LIN {X 0,Y 105.077,Z 582.031,A -85,B 0,C 180,E1 -30092.346,E2 -30092.346} C_VEL
LIN {X 0,Y 107.471,Z 573.639,A -85,B 0,C 180,E1 -30085.983,E2 -30085.983} C_VEL
LIN {X 0,Y 110.24,Z 565.564,A -85,B 0,C 180,E1 -30081.011,E2 -30081.011} C_VEL
LIN {X 0,Y 113.116,Z 557.316,A -85,B 0,C 180,E1 -30076.748,E2 -30076.748} C_VEL
LIN {X 0,Y 115.626,Z 549.926,A -85,B 0,C 180,E1 -30073.463,E2 -30073.463} C_VEL
LIN {X 0,Y 116.51,Z 546.107,A -85,B 0,C 180,E1 -30071.392,E2 -30071.392} C_VEL
LIN {X 0,Y 117.304,Z 542.305,A -85,B 0,C 180,E1 -30068.612,E2 -30068.612} C_VEL
LIN {X 0,Y 117.606,Z 540.558,A -85,B 0,C 180,E1 -30066.862,E2 -30066.862} C_VEL
LIN {X 0,Y 117.834,Z 538.313,A -85,B 0,C 180,E1 -30063.417,E2 -30063.417} C_VEL
LIN {X 0,Y 118.164,Z 536.971,A -85,B 0,C 180,E1 -30059.786,E2 -30059.786} C_VEL
LIN {X 0,Y 117.435,Z 539.078,A -85,B 0,C 180,E1 -30059.619,E2 -30059.619} C_VEL
LIN {X 0,Y 111.577,Z 552.371,A -85,B 0,C 180,E1 -30059.383,E2 -30059.383} C_VEL
LIN {X 0,Y 105.436,Z 562.957,A -85,B 0,C 180,E1 -30059.029,E2 -30059.029} C_VEL
LIN {X 0,Y 99.299,Z 571.677,A -85,B 0,C 180,E1 -30058.64,E2 -30058.64} C_VEL
LIN {X 0,Y 93.169,Z 579.093,A -85,B 0,C 180,E1 -30058.17,E2 -30058.17} C_VEL
LIN {X 0,Y 84.425,Z 587.882,A -85,B 0,C 180,E1 -30057.383,E2 -30057.383} C_VEL
LIN {X 0,Y 77.446,Z 593.868,A -85,B 0,C 180,E1 -30056.59,E2 -30056.59} C_VEL
LIN {X 0,Y 68.748,Z 600.175,A -85,B 0,C 180,E1 -30055.373,E2 -30055.373} C_VEL
LIN {X 0,Y 59.766,Z 605.63,A -85,B 0,C 180,E1 -30053.555,E2 -30053.555} C_VEL
LIN {X 0,Y 49.832,Z 610.547,A -85,B 0,C 180,E1 -30050.847,E2 -30050.847} C_VEL
LIN {X 0,Y 39.701,Z 614.514,A -85,B 0,C 180,E1 -30046.82,E2 -30046.82} C_VEL
LIN {X 0,Y 29.883,Z 617.454,A -85,B 0,C 180,E1 -30040.186,E2 -30040.186} C_VEL
LIN {X 0,Y 23.761,Z 618.964,A -85,B 0,C 180,E1 -30032.551,E2 -30032.551} C_VEL
LIN {X 0,Y 14.253,Z 620.512,A -85,B 0,C 180,E1 -29999.553,E2 -29999.553} C_VEL
LIN {X 0,Y 12.872,Z 620.802,A -85,B 0,C 180,E1 -29970.009,E2 -29970.009} C_VEL
LIN {X 0,Y 18.308,Z 619.905,A -85,B 0,C 180,E1 -29919.86,E2 -29919.86} C_VEL
LIN {X 0,Y 23.759,Z 618.965,A -85,B 0,C 180,E1 -29907.463,E2 -29907.463} C_VEL
LIN {X 0,Y 36.38,Z 615.606,A -85,B 0,C 180,E1 -29895.017,E2 -29895.017} C_VEL
LIN {X 0,Y 46.424,Z 611.976,A -85,B 0,C 180,E1 -29890.275,E2 -29890.275} C_VEL
LIN {X 0,Y 54.798,Z 608.214,A -85,B 0,C 180,E1 -29887.618,E2 -29887.618} C_VEL
LIN {X 0,Y 65.275,Z 602.361,A -85,B 0,C 180,E1 -29885.202,E2 -29885.202} C_VEL
LIN {X 0,Y 73.957,Z 596.492,A -85,B 0,C 180,E1 -29883.84,E2 -29883.84} C_VEL
LIN {X 0,Y 80.928,Z 591.003,A -85,B 0,C 180,E1 -29882.97,E2 -29882.97} C_VEL
LIN {X 0,Y 89.662,Z 582.792,A -85,B 0,C 180,E1 -29882.072,E2 -29882.072} C_VEL
LIN {X 0,Y 96.667,Z 574.974,A -85,B 0,C 180,E1 -29881.544,E2 -29881.544} C_VEL
LIN {X 0,Y 102.802,Z 566.899,A -85,B 0,C 180,E1 -29881.148,E2 -29881.148} C_VEL
LIN {X 0,Y 108.941,Z 557.148,A -85,B 0,C 180,E1 -29880.804,E2 -29880.804} C_VEL
LIN {X 0,Y 113.845,Z 547.604,A -85,B 0,C 180,E1 -29880.518,E2 -29880.518} C_VEL
LIN {X 0,Y 117.948,Z 537.604,A -85,B 0,C 180,E1 -29880.345,E2 -29880.345} C_VEL
LIN {X 0,Y 118.156,Z 536.995,A -85,B 0,C 180,E1 -29880.214,E2 -29880.214} C_VEL
LIN {X 0,Y 117.764,Z 538.933,A -85,B 0,C 180,E1 -29875.407,E2 -29875.407} C_VEL
LIN {X 0,Y 117.595,Z 540.587,A -85,B 0,C 180,E1 -29873.137,E2 -29873.137} C_VEL
LIN {X 0,Y 117.104,Z 543.335,A -85,B 0,C 180,E1 -29870.502,E2 -29870.502} C_VEL
LIN {X 0,Y 116.14,Z 547.81,A -85,B 0,C 180,E1 -29867.597,E2 -29867.597} C_VEL
LIN {X 0,Y 114.656,Z 552.807,A -85,B 0,C 180,E1 -29865.226,E2 -29865.226} C_VEL
LIN {X 0,Y 111.526,Z 561.914,A -85,B 0,C 180,E1 -29860.948,E2 -29860.948} C_VEL
LIN {X 0,Y 108.525,Z 570.445,A -85,B 0,C 180,E1 -29856.127,E2 -29856.127} C_VEL
LIN {X 0,Y 105.997,Z 578.44,A -85,B 0,C 180,E1 -29850.552,E2 -29850.552} C_VEL
LIN {X 0,Y 104.537,Z 584.513,A -85,B 0,C 180,E1 -29845.536,E2 -29845.536} C_VEL
LIN {X 0,Y 103.789,Z 592.504,A -85,B 0,C 180,E1 -29837.382,E2 -29837.382} C_VEL
LIN {X 0,Y 104.447,Z 596.825,A -85,B 0,C 180,E1 -29832.258,E2 -29832.258} C_VEL
LIN {X 0,Y 106.982,Z 602.173,A -85,B 0,C 180,E1 -29824.805,E2 -29824.805} C_VEL
LIN {X 0,Y 112.946,Z 607.538,A -85,B 0,C 180,E1 -29815.82,E2 -29815.82} C_VEL
LIN {X 0,Y 119.388,Z 610.725,A -85,B 0,C 180,E1 -29809.638,E2 -29809.638} C_VEL
LIN {X 0,Y 130.261,Z 613.684,A -85,B 0,C 180,E1 -29802.462,E2 -29802.462} C_VEL
LIN {X 0,Y 141.664,Z 615.261,A -85,B 0,C 180,E1 -29797.173,E2 -29797.173} C_VEL
LIN {X 0,Y 154.948,Z 615.935,A -85,B 0,C 180,E1 -29792.599,E2 -29792.599} C_VEL
LIN {X 0,Y 164.361,Z 615.933,A -85,B 0,C 180,E1 -29789.999,E2 -29789.999} C_VEL
LIN {X 0,Y 146.045,Z 615.598,A -85,B 0,C 180,E1 -29784.476,E2 -29784.476} C_VEL
LIN {X 0,Y 135.511,Z 614.596,A -85,B 0,C 180,E1 -29780.186,E2 -29780.186} C_VEL
LIN {X 0,Y 128.24,Z 613.248,A -85,B 0,C 180,E1 -29776.399,E2 -29776.399} C_VEL
LIN {X 0,Y 124.259,Z 612.62,A -85,B 0,C 180,E1 -29774.437,E2 -29774.437} C_VEL
LIN {X 0,Y 110.941,Z 610.999,A -85,B 0,C 180,E1 -29768.696,E2 -29768.696} C_VEL
LIN {X 0,Y 107.457,Z 610.024,A -85,B 0,C 180,E1 -29766.262,E2 -29766.262} C_VEL
LIN {X 0,Y 106.575,Z 609.586,A -85,B 0,C 180,E1 -29765.354,E2 -29765.354} C_VEL
LIN {X 0,Y 102.211,Z 606.637,A -85,B 0,C 180,E1 -29759.256,E2 -29759.256} C_VEL
LIN {X 0,Y 98.452,Z 601.21,A -85,B 0,C 180,E1 -29750.023,E2 -29750.023} C_VEL
LIN {X 0,Y 97.503,Z 596.13,A -85,B 0,C 180,E1 -29742.705,E2 -29742.705} C_VEL
LIN {X 0,Y 98.308,Z 589.496,A -85,B 0,C 180,E1 -29734.881,E2 -29734.881} C_VEL
LIN {X 0,Y 100.536,Z 582.409,A -85,B 0,C 180,E1 -29728.151,E2 -29728.151} C_VEL
LIN {X 0,Y 103.813,Z 574.191,A -85,B 0,C 180,E1 -29721.856,E2 -29721.856} C_VEL
LIN {X 0,Y 107.554,Z 565.572,A -85,B 0,C 180,E1 -29716.609,E2 -29716.609} C_VEL
LIN {X 0,Y 111.41,Z 556.493,A -85,B 0,C 180,E1 -29712.154,E2 -29712.154} C_VEL
LIN {X 0,Y 112.579,Z 553.533,A -85,B 0,C 180,E1 -29710.792,E2 -29710.792} C_VEL
LIN {X 0,Y 113.773,Z 550.19,A -85,B 0,C 180,E1 -29708.751,E2 -29708.751} C_VEL
LIN {X 0,Y 114.358,Z 547.971,A -85,B 0,C 180,E1 -29707.058,E2 -29707.058} C_VEL
LIN {X 0,Y 114.767,Z 546.299,A -85,B 0,C 180,E1 -29705.268,E2 -29705.268} C_VEL
LIN {X 0,Y 115.054,Z 545.147,A -85,B 0,C 180,E1 -29703.5,E2 -29703.5} C_VEL
LIN {X 0,Y 114.199,Z 546.967,A -85,B 0,C 180,E1 -29703.047,E2 -29703.047} C_VEL
LIN {X 0,Y 109.078,Z 556.945,A -85,B 0,C 180,E1 -29702.933,E2 -29702.933} C_VEL
LIN {X 0,Y 102.91,Z 566.698,A -85,B 0,C 180,E1 -29702.821,E2 -29702.821} C_VEL
LIN {X 0,Y 94.979,Z 576.963,A -85,B 0,C 180,E1 -29702.628,E2 -29702.628} C_VEL
LIN {X 0,Y 86.163,Z 586.127,A -85,B 0,C 180,E1 -29702.287,E2 -29702.287} C_VEL
LIN {X 0,Y 77.35,Z 593.672,A -85,B 0,C 180,E1 -29701.859,E2 -29701.859} C_VEL
LIN {X 0,Y 68.542,Z 599.979,A -85,B 0,C 180,E1 -29701.314,E2 -29701.314} C_VEL
LIN {X 0,Y 59.742,Z 605.253,A -85,B 0,C 180,E1 -29700.493,E2 -29700.493} C_VEL
LIN {X 0,Y 49.204,Z 610.351,A -85,B 0,C 180,E1 -29699.077,E2 -29699.077} C_VEL
LIN {X 0,Y 38.703,Z 614.318,A -85,B 0,C 180,E1 -29697.167,E2 -29697.167} C_VEL
LIN {X 0,Y 28.274,Z 617.258,A -85,B 0,C 180,E1 -29693.896,E2 -29693.896} C_VEL
LIN {X 0,Y 21.426,Z 618.768,A -85,B 0,C 180,E1 -29689.771,E2 -29689.771} C_VEL
LIN {X 0,Y 8.797,Z 620.316,A -85,B 0,C 180,E1 -29663.046,E2 -29663.046} C_VEL
LIN {X 0,Y 5.76,Z 620.606,A -85,B 0,C 180,E1 -29610.021,E2 -29610.021} C_VEL
LIN {X 0,Y 14.789,Z 619.709,A -85,B 0,C 180,E1 -29538.142,E2 -29538.142} C_VEL
LIN {X 0,Y 21.423,Z 618.769,A -85,B 0,C 180,E1 -29530.243,E2 -29530.243} C_VEL
LIN {X 0,Y 35.213,Z 615.41,A -85,B 0,C 180,E1 -29523.759,E2 -29523.759} C_VEL
LIN {X 0,Y 45.694,Z 611.781,A -85,B 0,C 180,E1 -29521.46,E2 -29521.46} C_VEL
LIN {X 0,Y 56.221,Z 607.046,A -85,B 0,C 180,E1 -29519.891,E2 -29519.891} C_VEL
LIN {X 0,Y 66.778,Z 601.073,A -85,B 0,C 180,E1 -29518.785,E2 -29518.785} C_VEL
LIN {X 0,Y 75.586,Z 594.984,A -85,B 0,C 180,E1 -29518.188,E2 -29518.188} C_VEL
LIN {X 0,Y 82.634,Z 589.249,A -85,B 0,C 180,E1 -29517.849,E2 -29517.849} C_VEL
LIN {X 0,Y 89.687,Z 582.597,A -85,B 0,C 180,E1 -29517.53,E2 -29517.53} C_VEL
LIN {X 0,Y 96.736,Z 574.78,A -85,B 0,C 180,E1 -29517.338,E2 -29517.338} C_VEL
LIN {X 0,Y 102.905,Z 566.704,A -85,B 0,C 180,E1 -29517.189,E2 -29517.189} C_VEL
LIN {X 0,Y 109.072,Z 556.953,A -85,B 0,C 180,E1 -29517.076,E2 -29517.076} C_VEL
LIN {X 0,Y 114.158,Z 547.059,A -85,B 0,C 180,E1 -29516.952,E2 -29516.952} C_VEL
LIN {X 0,Y 115.07,Z 545.112,A -85,B 0,C 180,E1 -29516.5,E2 -29516.5} C_VEL
LIN {X 0,Y 114.759,Z 546.317,A -85,B 0,C 180,E1 -29514.731,E2 -29514.731} C_VEL
LIN {X 0,Y 114.117,Z 548.954,A -85,B 0,C 180,E1 -29512.089,E2 -29512.089} C_VEL
LIN {X 0,Y 112.59,Z 553.513,A -85,B 0,C 180,E1 -29509.209,E2 -29509.209} C_VEL
LIN {X 0,Y 108.961,Z 562.356,A -85,B 0,C 180,E1 -29505.051,E2 -29505.051} C_VEL
LIN {X 0,Y 105.384,Z 570.543,A -85,B 0,C 180,E1 -29500.524,E2 -29500.524} C_VEL
LIN {X 0,Y 102.338,Z 577.72,A -85,B 0,C 180,E1 -29495.669,E2 -29495.669} C_VEL
LIN {X 0,Y 99.681,Z 584.762,A -85,B 0,C 180,E1 -29489.842,E2 -29489.842} C_VEL
LIN {X 0,Y 97.81,Z 592.098,A -85,B 0,C 180,E1 -29482.219,E2 -29482.219} C_VEL
LIN {X 0,Y 97.691,Z 598.503,A -85,B 0,C 180,E1 -29473.998,E2 -29473.998} C_VEL
LIN {X 0,Y 99.573,Z 603.51,A -85,B 0,C 180,E1 -29466.232,E2 -29466.232} C_VEL
LIN {X 0,Y 103.762,Z 607.822,A -85,B 0,C 180,E1 -29458.301,E2 -29458.301} C_VEL
LIN {X 0,Y 108.038,Z 610.419,A -85,B 0,C 180,E1 -29452.972,E2 -29452.972} C_VEL
LIN {X 0,Y 116.685,Z 613.42,A -85,B 0,C 180,E1 -29445.496,E2 -29445.496} C_VEL
LIN {X 0,Y 128.033,Z 615.375,A -85,B 0,C 180,E1 -29438.878,E2 -29438.878} C_VEL
LIN {X 0,Y 143.113,Z 616.254,A -85,B 0,C 180,E1 -29432.814,E2 -29432.814} C_VEL
LIN {X 0,Y 152.408,Z 616.261,A -85,B 0,C 180,E1 -29429.999,E2 -29429.999} C_VEL
LIN {X 0,Y 140.833,Z 616.242,A -85,B 0,C 180,E1 -29426.403,E2 -29426.403} C_VEL
LIN {X 0,Y 126.578,Z 615.235,A -85,B 0,C 180,E1 -29420.411,E2 -29420.411} C_VEL
LIN {X 0,Y 116.686,Z 613.419,A -85,B 0,C 180,E1 -29414.503,E2 -29414.503} C_VEL
LIN {X 0,Y 106.575,Z 609.586,A -85,B 0,C 180,E1 -29405.354,E2 -29405.354} C_VEL
LIN {X 0,Y 103.743,Z 608.404,A -85,B 0,C 180,E1 -29402.603,E2 -29402.603} C_VEL
LIN {X 0,Y 94.034,Z 605.542,A -85,B 0,C 180,E1 -29394.078,E2 -29394.078} C_VEL
LIN {X 0,Y 92.077,Z 604.091,A -85,B 0,C 180,E1 -29390.778,E2 -29390.778} C_VEL
LIN {X 0,Y 91.753,Z 603.497,A -85,B 0,C 180,E1 -29389.63,E2 -29389.63} C_VEL
LIN {X 0,Y 91.292,Z 597.32,A -85,B 0,C 180,E1 -29379.659,E2 -29379.659} C_VEL
LIN {X 0,Y 93.298,Z 590.008,A -85,B 0,C 180,E1 -29370.557,E2 -29370.557} C_VEL
LIN {X 0,Y 96.591,Z 582.776,A -85,B 0,C 180,E1 -29363.585,E2 -29363.585} C_VEL
LIN {X 0,Y 100.516,Z 575.187,A -85,B 0,C 180,E1 -29357.754,E2 -29357.754} C_VEL
LIN {X 0,Y 104.996,Z 566.701,A -85,B 0,C 180,E1 -29352.635,E2 -29352.635} C_VEL
LIN {X 0,Y 109.261,Z 558.245,A -85,B 0,C 180,E1 -29348.527,E2 -29348.527} C_VEL
LIN {X 0,Y 110.195,Z 556.06,A -85,B 0,C 180,E1 -29347.326,E2 -29347.326} C_VEL
LIN {X 0,Y 109.153,Z 557.682,A -85,B 0,C 180,E1 -29346.649,E2 -29346.649} C_VEL
LIN {X 0,Y 101.74,Z 569.068,A -85,B 0,C 180,E1 -29346.783,E2 -29346.783} C_VEL
LIN {X 0,Y 93.801,Z 578.702,A -85,B 0,C 180,E1 -29346.901,E2 -29346.901} C_VEL
LIN {X 0,Y 84.975,Z 587.49,A -85,B 0,C 180,E1 -29347.027,E2 -29347.027} C_VEL
LIN {X 0,Y 77.908,Z 593.476,A -85,B 0,C 180,E1 -29347.111,E2 -29347.111} C_VEL
LIN {X 0,Y 69.075,Z 599.783,A -85,B 0,C 180,E1 -29347.24,E2 -29347.24} C_VEL
LIN {X 0,Y 60.227,Z 605.057,A -85,B 0,C 180,E1 -29347.299,E2 -29347.299} C_VEL
LIN {X 0,Y 49.605,Z 610.155,A -85,B 0,C 180,E1 -29347.346,E2 -29347.346} C_VEL
LIN {X 0,Y 39.009,Z 614.121,A -85,B 0,C 180,E1 -29347.715,E2 -29347.715} C_VEL
LIN {X 0,Y 28.413,Z 617.063,A -85,B 0,C 180,E1 -29348.319,E2 -29348.319} C_VEL
LIN {X 0,Y 21.349,Z 618.572,A -85,B 0,C 180,E1 -29349.001,E2 -29349.001} C_VEL
LIN {X 0,Y 7.268,Z 620.121,A -85,B 0,C 180,E1 -29354.692,E2 -29354.692} C_VEL
LIN {X 0,Y 1.339,Z 620.411,A -85,B 0,C 180,E1 -29429.911,E2 -29429.911} C_VEL
LIN {X 0,Y 14.281,Z 619.512,A -85,B 0,C 180,E1 -29509.759,E2 -29509.759} C_VEL
LIN {X 0,Y 21.344,Z 618.572,A -85,B 0,C 180,E1 -29511.009,E2 -29511.009} C_VEL
LIN {X 0,Y 35.465,Z 615.215,A -85,B 0,C 180,E1 -29512.207,E2 -29512.207} C_VEL
LIN {X 0,Y 46.065,Z 611.585,A -85,B 0,C 180,E1 -29512.577,E2 -29512.577} C_VEL
LIN {X 0,Y 54.75,Z 607.83,A -85,B 0,C 180,E1 -29512.629,E2 -29512.629} C_VEL
LIN {X 0,Y 65.541,Z 601.969,A -85,B 0,C 180,E1 -29512.675,E2 -29512.675} C_VEL
LIN {X 0,Y 74.377,Z 596.1,A -85,B 0,C 180,E1 -29512.802,E2 -29512.802} C_VEL
LIN {X 0,Y 81.44,Z 590.612,A -85,B 0,C 180,E1 -29512.918,E2 -29512.918} C_VEL
LIN {X 0,Y 90.272,Z 582.402,A -85,B 0,C 180,E1 -29513.022,E2 -29513.022} C_VEL
LIN {X 0,Y 97.324,Z 574.585,A -85,B 0,C 180,E1 -29513.163,E2 -29513.163} C_VEL
LIN {X 0,Y 103.5,Z 566.508,A -85,B 0,C 180,E1 -29513.243,E2 -29513.243} C_VEL
LIN {X 0,Y 109.165,Z 557.66,A -85,B 0,C 180,E1 -29513.352,E2 -29513.352} C_VEL
LIN {X 0,Y 110.209,Z 556.036,A -85,B 0,C 180,E1 -29512.675,E2 -29512.675} C_VEL
LIN {X 0,Y 108.123,Z 560.659,A -85,B 0,C 180,E1 -29510.358,E2 -29510.358} C_VEL
LIN {X 0,Y 102.874,Z 570.73,A -85,B 0,C 180,E1 -29505.055,E2 -29505.055} C_VEL
LIN {X 0,Y 99.18,Z 577.737,A -85,B 0,C 180,E1 -29500.46,E2 -29500.46} C_VEL
LIN {X 0,Y 95.041,Z 585.875,A -85,B 0,C 180,E1 -29493.664,E2 -29493.664} C_VEL
LIN {X 0,Y 92.415,Z 592.353,A -85,B 0,C 180,E1 -29486.773,E2 -29486.773} C_VEL
LIN {X 0,Y 91.133,Z 598.33,A -85,B 0,C 180,E1 -29478.824,E2 -29478.824} C_VEL
LIN {X 0,Y 91.814,Z 603.668,A -85,B 0,C 180,E1 -29470.056,E2 -29470.056} C_VEL
LIN {X 0,Y 94.928,Z 608.101,A -85,B 0,C 180,E1 -29461.213,E2 -29461.213} C_VEL
LIN {X 0,Y 99.815,Z 611.279,A -85,B 0,C 180,E1 -29453.753,E2 -29453.753} C_VEL
LIN {X 0,Y 109.068,Z 614.307,A -85,B 0,C 180,E1 -29444.87,E2 -29444.87} C_VEL
LIN {X 0,Y 115.689,Z 615.539,A -85,B 0,C 180,E1 -29440.5,E2 -29440.5} C_VEL
LIN {X 0,Y 126.957,Z 616.51,A -85,B 0,C 180,E1 -29434.864,E2 -29434.864} C_VEL
LIN {X 0,Y 140.502,Z 616.589,A -85,B 0,C 180,E1 -29429.999,E2 -29429.999} C_VEL
LIN {X 0,Y 126.957,Z 616.511,A -85,B 0,C 180,E1 -29425.137,E2 -29425.137} C_VEL
LIN {X 0,Y 114.603,Z 615.378,A -85,B 0,C 180,E1 -29418.861,E2 -29418.861} C_VEL
LIN {X 0,Y 103.318,Z 612.677,A -85,B 0,C 180,E1 -29410.115,E2 -29410.115} C_VEL
LIN {X 0,Y 98.607,Z 610.701,A -85,B 0,C 180,E1 -29404.681,E2 -29404.681} C_VEL
LIN {X 0,Y 93.548,Z 606.716,A -85,B 0,C 180,E1 -29395.726,E2 -29395.726} C_VEL
LIN {X 0,Y 91.753,Z 603.497,A -85,B 0,C 180,E1 -29389.63,E2 -29389.63} C_VEL
LIN {X 0,Y 90.644,Z 601.814,A -85,B 0,C 180,E1 -29386.132,E2 -29386.132} C_VEL
LIN {X 0,Y 86.492,Z 597.323,A -85,B 0,C 180,E1 -29375.271,E2 -29375.271} C_VEL
LIN {X 0,Y 86.524,Z 595.201,A -85,B 0,C 180,E1 -29371.632,E2 -29371.632} C_VEL
LIN {X 0,Y 86.848,Z 594.361,A -85,B 0,C 180,E1 -29370.479,E2 -29370.479} C_VEL
LIN {X 0,Y 89.45,Z 589.522,A -85,B 0,C 180,E1 -29364.804,E2 -29364.804} C_VEL
LIN {X 0,Y 93.187,Z 583.394,A -85,B 0,C 180,E1 -29358.914,E2 -29358.914} C_VEL
LIN {X 0,Y 97.785,Z 576.195,A -85,B 0,C 180,E1 -29353.476,E2 -29353.476} C_VEL
LIN {X 0,Y 100.185,Z 572.189,A -85,B 0,C 180,E1 -29350.855,E2 -29350.855} C_VEL
LIN {X 0,Y 93.164,Z 580.355,A -85,B 0,C 180,E1 -29351.279,E2 -29351.279} C_VEL
LIN {X 0,Y 86.137,Z 587.294,A -85,B 0,C 180,E1 -29351.734,E2 -29351.734} C_VEL
LIN {X 0,Y 79.107,Z 593.281,A -85,B 0,C 180,E1 -29352.238,E2 -29352.238} C_VEL
LIN {X 0,Y 70.328,Z 599.588,A -85,B 0,C 180,E1 -29353.006,E2 -29353.006} C_VEL
LIN {X 0,Y 61.543,Z 604.861,A -85,B 0,C 180,E1 -29353.905,E2 -29353.905} C_VEL
LIN {X 0,Y 51.014,Z 609.959,A -85,B 0,C 180,E1 -29355.335,E2 -29355.335} C_VEL
LIN {X 0,Y 40.589,Z 613.925,A -85,B 0,C 180,E1 -29357.757,E2 -29357.757} C_VEL
LIN {X 0,Y 30.271,Z 616.868,A -85,B 0,C 180,E1 -29361.762,E2 -29361.762} C_VEL
LIN {X 0,Y 23.547,Z 618.375,A -85,B 0,C 180,E1 -29366.432,E2 -29366.432} C_VEL
LIN {X 0,Y 11.394,Z 619.925,A -85,B 0,C 180,E1 -29391.902,E2 -29391.902} C_VEL
LIN {X 0,Y 8.43,Z 620.217,A -85,B 0,C 180,E1 -29429.986,E2 -29429.986} C_VEL
LIN {X 0,Y 17.063,Z 619.316,A -85,B 0,C 180,E1 -29485.451,E2 -29485.451} C_VEL
LIN {X 0,Y 23.542,Z 618.376,A -85,B 0,C 180,E1 -29493.574,E2 -29493.574} C_VEL
LIN {X 0,Y 37.113,Z 615.019,A -85,B 0,C 180,E1 -29501.221,E2 -29501.221} C_VEL
LIN {X 0,Y 47.512,Z 611.39,A -85,B 0,C 180,E1 -29504.033,E2 -29504.033} C_VEL
LIN {X 0,Y 58.031,Z 606.654,A -85,B 0,C 180,E1 -29505.651,E2 -29505.651} C_VEL
LIN {X 0,Y 68.582,Z 600.68,A -85,B 0,C 180,E1 -29506.775,E2 -29506.775} C_VEL
LIN {X 0,Y 77.354,Z 594.594,A -85,B 0,C 180,E1 -29507.595,E2 -29507.595} C_VEL
LIN {X 0,Y 84.379,Z 588.857,A -85,B 0,C 180,E1 -29508.134,E2 -29508.134} C_VEL
LIN {X 0,Y 91.407,Z 582.207,A -85,B 0,C 180,E1 -29508.601,E2 -29508.601} C_VEL
LIN {X 0,Y 98.426,Z 574.389,A -85,B 0,C 180,E1 -29509.043,E2 -29509.043} C_VEL
LIN {X 0,Y 100.181,Z 572.194,A -85,B 0,C 180,E1 -29509.144,E2 -29509.144} C_VEL
LIN {X 0,Y 100.239,Z 572.186,A -85,B 0,C 180,E1 -29508.973,E2 -29508.973} C_VEL
LIN {X 0,Y 95.876,Z 579.075,A -85,B 0,C 180,E1 -29504.505,E2 -29504.505} C_VEL
LIN {X 0,Y 90.994,Z 586.841,A -85,B 0,C 180,E1 -29497.941,E2 -29497.941} C_VEL
LIN {X 0,Y 87.5,Z 593.057,A -85,B 0,C 180,E1 -29491.192,E2 -29491.192} C_VEL
LIN {X 0,Y 85.18,Z 598.78,A -85,B 0,C 180,E1 -29483.272,E2 -29483.272} C_VEL
LIN {X 0,Y 84.56,Z 603.57,A -85,B 0,C 180,E1 -29475.056,E2 -29475.056} C_VEL
LIN {X 0,Y 86.476,Z 608.378,A -85,B 0,C 180,E1 -29464.671,E2 -29464.671} C_VEL
LIN {X 0,Y 89.423,Z 610.985,A -85,B 0,C 180,E1 -29458.134,E2 -29458.134} C_VEL
LIN {X 0,Y 98.728,Z 614.577,A -85,B 0,C 180,E1 -29446.542,E2 -29446.542} C_VEL
LIN {X 0,Y 107.09,Z 616.069,A -85,B 0,C 180,E1 -29440.144,E2 -29440.144} C_VEL
LIN {X 0,Y 120.072,Z 616.879,A -85,B 0,C 180,E1 -29433.355,E2 -29433.355} C_VEL
LIN {X 0,Y 128.829,Z 616.909,A -85,B 0,C 180,E1 -29429.999,E2 -29429.999} C_VEL
LIN {X 0,Y 113.198,Z 616.623,A -85,B 0,C 180,E1 -29423.381,E2 -29423.381} C_VEL
LIN {X 0,Y 104.929,Z 615.84,A -85,B 0,C 180,E1 -29418.407,E2 -29418.407} C_VEL
LIN {X 0,Y 96.496,Z 614.025,A -85,B 0,C 180,E1 -29411.222,E2 -29411.222} C_VEL
LIN {X 0,Y 88.735,Z 610.478,A -85,B 0,C 180,E1 -29400.596,E2 -29400.596} C_VEL
LIN {X 0,Y 85.071,Z 605.848,A -85,B 0,C 180,E1 -29389.654,E2 -29389.654} C_VEL
LIN {X 0,Y 84.601,Z 601.739,A -85,B 0,C 180,E1 -29381.612,E2 -29381.612} C_VEL
LIN {X 0,Y 86.378,Z 595.405,A -85,B 0,C 180,E1 -29371.832,E2 -29371.832} C_VEL
LIN {X 0,Y 86.848,Z 594.361,A -85,B 0,C 180,E1 -29370.479,E2 -29370.479} C_VEL
LIN {X 0,Y 87.21,Z 592.877,A -85,B 0,C 180,E1 -29368.052,E2 -29368.052} C_VEL
LIN {X 0,Y 86.672,Z 589.315,A -85,B 0,C 180,E1 -29359.468,E2 -29359.468} C_VEL
LIN {X 0,Y 87.679,Z 587.578,A -85,B 0,C 180,E1 -29357.208,E2 -29357.208} C_VEL
LIN {X 0,Y 88.062,Z 587.079,A -85,B 0,C 180,E1 -29356.725,E2 -29356.725} C_VEL
LIN {X 0,Y 87.863,Z 587.099,A -85,B 0,C 180,E1 -29356.287,E2 -29356.287} C_VEL
LIN {X 0,Y 80.915,Z 593.085,A -85,B 0,C 180,E1 -29357.169,E2 -29357.169} C_VEL
LIN {X 0,Y 72.27,Z 599.391,A -85,B 0,C 180,E1 -29358.528,E2 -29358.528} C_VEL
LIN {X 0,Y 63.639,Z 604.665,A -85,B 0,C 180,E1 -29360.162,E2 -29360.162} C_VEL
LIN {X 0,Y 53.35,Z 609.763,A -85,B 0,C 180,E1 -29362.754,E2 -29362.754} C_VEL
LIN {X 0,Y 43.301,Z 613.729,A -85,B 0,C 180,E1 -29366.783,E2 -29366.783} C_VEL
LIN {X 0,Y 33.563,Z 616.672,A -85,B 0,C 180,E1 -29373.109,E2 -29373.109} C_VEL
LIN {X 0,Y 27.479,Z 618.179,A -85,B 0,C 180,E1 -29379.883,E2 -29379.883} C_VEL
LIN {X 0,Y 17.55,Z 619.729,A -85,B 0,C 180,E1 -29406.386,E2 -29406.386} C_VEL
LIN {X 0,Y 15.539,Z 620.021,A -85,B 0,C 180,E1 -29429.992,E2 -29429.992} C_VEL
LIN {X 0,Y 21.908,Z 619.121,A -85,B 0,C 180,E1 -29469.904,E2 -29469.904} C_VEL
LIN {X 0,Y 27.473,Z 618.18,A -85,B 0,C 180,E1 -29480.118,E2 -29480.118} C_VEL
LIN {X 0,Y 39.992,Z 614.822,A -85,B 0,C 180,E1 -29491.475,E2 -29491.475} C_VEL
LIN {X 0,Y 49.953,Z 611.194,A -85,B 0,C 180,E1 -29496.128,E2 -29496.128} C_VEL
LIN {X 0,Y 56.478,Z 608.401,A -85,B 0,C 180,E1 -29498.084,E2 -29498.084} C_VEL
LIN {X 0,Y 67.101,Z 602.669,A -85,B 0,C 180,E1 -29500.492,E2 -29500.492} C_VEL
LIN {X 0,Y 75.732,Z 597.019,A -85,B 0,C 180,E1 -29502.022,E2 -29502.022} C_VEL
LIN {X 0,Y 84.381,Z 590.222,A -85,B 0,C 180,E1 -29503.293,E2 -29503.293} C_VEL
LIN {X 0,Y 87.865,Z 587.102,A -85,B 0,C 180,E1 -29503.7,E2 -29503.7} C_VEL
LIN {X 0,Y 88.042,Z 587.085,A -85,B 0,C 180,E1 -29503.309,E2 -29503.309} C_VEL
LIN {X 0,Y 83.839,Z 592.853,A -85,B 0,C 180,E1 -29497.23,E2 -29497.23} C_VEL
LIN {X 0,Y 79.786,Z 599.352,A -85,B 0,C 180,E1 -29488.098,E2 -29488.098} C_VEL
LIN {X 0,Y 77.999,Z 604.463,A -85,B 0,C 180,E1 -29478.626,E2 -29478.626} C_VEL
LIN {X 0,Y 78.577,Z 608.648,A -85,B 0,C 180,E1 -29468.759,E2 -29468.759} C_VEL
LIN {X 0,Y 81.237,Z 611.69,A -85,B 0,C 180,E1 -29460.109,E2 -29460.109} C_VEL
LIN {X 0,Y 88.842,Z 614.895,A -85,B 0,C 180,E1 -29448.336,E2 -29448.336} C_VEL
LIN {X 0,Y 94.447,Z 616.135,A -85,B 0,C 180,E1 -29442.898,E2 -29442.898} C_VEL
LIN {X 0,Y 108.888,Z 617.186,A -85,B 0,C 180,E1 -29433.699,E2 -29433.699} C_VEL
LIN {X 0,Y 117.322,Z 617.225,A -85,B 0,C 180,E1 -29429.999,E2 -29429.999} C_VEL
LIN {X 0,Y 105.861,Z 617.161,A -85,B 0,C 180,E1 -29424.74,E2 -29424.74} C_VEL
LIN {X 0,Y 93.907,Z 616.041,A -85,B 0,C 180,E1 -29416.625,E2 -29416.625} C_VEL
LIN {X 0,Y 84.064,Z 613.248,A -85,B 0,C 180,E1 -29405.289,E2 -29405.289} C_VEL
LIN {X 0,Y 80.631,Z 611.262,A -85,B 0,C 180,E1 -29398.467,E2 -29398.467} C_VEL
LIN {X 0,Y 77.971,Z 606.616,A -85,B 0,C 180,E1 -29386.14,E2 -29386.14} C_VEL
LIN {X 0,Y 78.696,Z 601.996,A -85,B 0,C 180,E1 -29376.508,E2 -29376.508} C_VEL
LIN {X 0,Y 81.21,Z 596.903,A -85,B 0,C 180,E1 -29368.095,E2 -29368.095} C_VEL
LIN {X 0,Y 86.328,Z 589.404,A -85,B 0,C 180,E1 -29359.002,E2 -29359.002} C_VEL
LIN {X 0,Y 87.679,Z 587.578,A -85,B 0,C 180,E1 -29357.208,E2 -29357.208} C_VEL
LIN {X 0,Y 87.234,Z 587.83,A -85,B 0,C 180,E1 -29356.829,E2 -29356.829} C_VEL
LIN {X 0,Y 85.458,Z 589.332,A -85,B 0,C 180,E1 -29356.798,E2 -29356.798} C_VEL
LIN {X 0,Y 81.9,Z 592.565,A -85,B 0,C 180,E1 -29357.826,E2 -29357.826} C_VEL
LIN {X 0,Y 73.121,Z 599.858,A -85,B 0,C 180,E1 -29362.52,E2 -29362.52} C_VEL
LIN {X 0,Y 68.023,Z 603.515,A -85,B 0,C 180,E1 -29365.175,E2 -29365.175} C_VEL
LIN {X 0,Y 64.63,Z 605.434,A -85,B 0,C 180,E1 -29366.485,E2 -29366.485} C_VEL
LIN {X 0,Y 56.491,Z 609.567,A -85,B 0,C 180,E1 -29369.438,E2 -29369.438} C_VEL
LIN {X 0,Y 46.944,Z 613.534,A -85,B 0,C 180,E1 -29374.57,E2 -29374.57} C_VEL
LIN {X 0,Y 37.937,Z 616.476,A -85,B 0,C 180,E1 -29382.178,E2 -29382.178} C_VEL
LIN {X 0,Y 32.518,Z 617.983,A -85,B 0,C 180,E1 -29389.577,E2 -29389.577} C_VEL
LIN {X 0,Y 24.258,Z 619.533,A -85,B 0,C 180,E1 -29413.154,E2 -29413.154} C_VEL
LIN {X 0,Y 22.638,Z 619.826,A -85,B 0,C 180,E1 -29429.995,E2 -29429.995} C_VEL
LIN {X 0,Y 27.75,Z 618.925,A -85,B 0,C 180,E1 -29460.427,E2 -29460.427} C_VEL
LIN {X 0,Y 32.512,Z 617.984,A -85,B 0,C 180,E1 -29470.423,E2 -29470.423} C_VEL
LIN {X 0,Y 43.857,Z 614.626,A -85,B 0,C 180,E1 -29483.244,E2 -29483.244} C_VEL
LIN {X 0,Y 53.245,Z 610.997,A -85,B 0,C 180,E1 -29489.083,E2 -29489.083} C_VEL
LIN {X 0,Y 60.841,Z 607.482,A -85,B 0,C 180,E1 -29492.218,E2 -29492.218} C_VEL
LIN {X 0,Y 71.625,Z 601.291,A -85,B 0,C 180,E1 -29495.451,E2 -29495.451} C_VEL
LIN {X 0,Y 76.6,Z 598.086,A -85,B 0,C 180,E1 -29496.556,E2 -29496.556} C_VEL
LIN {X 0,Y 72.927,Z 603.28,A -85,B 0,C 180,E1 -29487.459,E2 -29487.459} C_VEL
LIN {X 0,Y 71.223,Z 608.916,A -85,B 0,C 180,E1 -29473.685,E2 -29473.685} C_VEL
LIN {X 0,Y 72.382,Z 611.535,A -85,B 0,C 180,E1 -29465.63,E2 -29465.63} C_VEL
LIN {X 0,Y 76.968,Z 614.526,A -85,B 0,C 180,E1 -29454.069,E2 -29454.069} C_VEL
LIN {X 0,Y 86.347,Z 616.688,A -85,B 0,C 180,E1 -29442.404,E2 -29442.404} C_VEL
LIN {X 0,Y 97.847,Z 617.49,A -85,B 0,C 180,E1 -29434.118,E2 -29434.118} C_VEL
LIN {X 0,Y 106.06,Z 617.535,A -85,B 0,C 180,E1 -29429.999,E2 -29429.999} C_VEL
LIN {X 0,Y 90.55,Z 617.124,A -85,B 0,C 180,E1 -29421.069,E2 -29421.069} C_VEL
LIN {X 0,Y 81.233,Z 615.735,A -85,B 0,C 180,E1 -29412.107,E2 -29412.107} C_VEL
LIN {X 0,Y 74.949,Z 613.527,A -85,B 0,C 180,E1 -29402.039,E2 -29402.039} C_VEL
LIN {X 0,Y 71.777,Z 610.63,A -85,B 0,C 180,E1 -29391.56,E2 -29391.56} C_VEL
LIN {X 0,Y 71.4,Z 606.741,A -85,B 0,C 180,E1 -29380.474,E2 -29380.474} C_VEL
LIN {X 0,Y 73.5,Z 602.254,A -85,B 0,C 180,E1 -29370.617,E2 -29370.617} C_VEL
LIN {X 0,Y 76.517,Z 598.089,A -85,B 0,C 180,E1 -29363.292,E2 -29363.292} C_VEL
LIN {X 0,Y 66.428,Z 604.47,A -85,B 0,C 180,E1 -29365.933,E2 -29365.933} C_VEL
LIN {X 0,Y 64.63,Z 605.434,A -85,B 0,C 180,E1 -29366.485,E2 -29366.485} C_VEL
LIN {X 0,Y 59.918,Z 608.132,A -85,B 0,C 180,E1 -29368.792,E2 -29368.792} C_VEL
LIN {X 0,Y 50.838,Z 613.044,A -85,B 0,C 180,E1 -29378.471,E2 -29378.471} C_VEL
LIN {X 0,Y 45.996,Z 615.317,A -85,B 0,C 180,E1 -29385.41,E2 -29385.41} C_VEL
LIN {X 0,Y 43.332,Z 616.181,A -85,B 0,C 180,E1 -29388.89,E2 -29388.89} C_VEL
LIN {X 0,Y 38.232,Z 617.787,A -85,B 0,C 180,E1 -29396.528,E2 -29396.528} C_VEL
LIN {X 0,Y 31.145,Z 619.338,A -85,B 0,C 180,E1 -29416.955,E2 -29416.955} C_VEL
LIN {X 0,Y 29.753,Z 619.631,A -85,B 0,C 180,E1 -29429.996,E2 -29429.996} C_VEL
LIN {X 0,Y 34.095,Z 618.729,A -85,B 0,C 180,E1 -29454.343,E2 -29454.343} C_VEL
LIN {X 0,Y 38.226,Z 617.788,A -85,B 0,C 180,E1 -29463.47,E2 -29463.47} C_VEL
LIN {X 0,Y 48.469,Z 614.43,A -85,B 0,C 180,E1 -29476.464,E2 -29476.464} C_VEL
LIN {X 0,Y 57.241,Z 610.801,A -85,B 0,C 180,E1 -29482.941,E2 -29482.941} C_VEL
LIN {X 0,Y 61.599,Z 608.8,A -85,B 0,C 180,E1 -29485.222,E2 -29485.222} C_VEL
LIN {X 0,Y 65.716,Z 606.947,A -85,B 0,C 180,E1 -29485.91,E2 -29485.91} C_VEL
LIN {X 0,Y 64.673,Z 611.865,A -85,B 0,C 180,E1 -29470.48,E2 -29470.48} C_VEL
LIN {X 0,Y 69.338,Z 615.373,A -85,B 0,C 180,E1 -29454.193,E2 -29454.193} C_VEL
LIN {X 0,Y 74.207,Z 616.71,A -85,B 0,C 180,E1 -29446.504,E2 -29446.504} C_VEL
LIN {X 0,Y 87.017,Z 617.789,A -85,B 0,C 180,E1 -29434.631,E2 -29434.631} C_VEL
LIN {X 0,Y 94.966,Z 617.839,A -85,B 0,C 180,E1 -29429.999,E2 -29429.999} C_VEL
LIN {X 0,Y 84.827,Z 617.764,A -85,B 0,C 180,E1 -29423.806,E2 -29423.806} C_VEL
LIN {X 0,Y 73.601,Z 616.591,A -85,B 0,C 180,E1 -29412.712,E2 -29412.712} C_VEL
LIN {X 0,Y 66.268,Z 613.802,A -85,B 0,C 180,E1 -29397.974,E2 -29397.974} C_VEL
LIN {X 0,Y 64.653,Z 611.804,A -85,B 0,C 180,E1 -29389.289,E2 -29389.289} C_VEL
LIN {X 0,Y 65.732,Z 606.94,A -85,B 0,C 180,E1 -29374.089,E2 -29374.089} C_VEL
LIN {X 0,Y 62.392,Z 608.4,A -85,B 0,C 180,E1 -29374.274,E2 -29374.274} C_VEL
LIN {X 0,Y 54.218,Z 612.214,A -85,B 0,C 180,E1 -29378.943,E2 -29378.943} C_VEL
LIN {X 0,Y 43.332,Z 616.181,A -85,B 0,C 180,E1 -29388.89,E2 -29388.89} C_VEL
LIN {X 0,Y 39.72,Z 617.5,A -85,B 0,C 180,E1 -29395.082,E2 -29395.082} C_VEL
LIN {X 0,Y 37.383,Z 618.466,A -85,B 0,C 180,E1 -29403.065,E2 -29403.065} C_VEL
LIN {X 0,Y 36.237,Z 619.395,A -85,B 0,C 180,E1 -29421.625,E2 -29421.625} C_VEL
LIN {X 0,Y 37.172,Z 619.327,A -85,B 0,C 180,E1 -29434.028,E2 -29434.028} C_VEL
LIN {X 0,Y 40.696,Z 618.533,A -85,B 0,C 180,E1 -29450.202,E2 -29450.202} C_VEL
LIN {X 0,Y 44.35,Z 617.592,A -85,B 0,C 180,E1 -29458.382,E2 -29458.382} C_VEL
LIN {X 0,Y 53.635,Z 614.234,A -85,B 0,C 180,E1 -29470.929,E2 -29470.929} C_VEL
LIN {X 0,Y 57.601,Z 612.926,A -85,B 0,C 180,E1 -29472.946,E2 -29472.946} C_VEL
LIN {X 0,Y 60.416,Z 615.708,A -85,B 0,C 180,E1 -29457.728,E2 -29457.728} C_VEL
LIN {X 0,Y 65.995,Z 617.229,A -85,B 0,C 180,E1 -29446.591,E2 -29446.591} C_VEL
LIN {X 0,Y 76.4,Z 618.082,A -85,B 0,C 180,E1 -29435.276,E2 -29435.276} C_VEL
LIN {X 0,Y 84.038,Z 618.14,A -85,B 0,C 180,E1 -29429.999,E2 -29429.999} C_VEL
LIN {X 0,Y 69.853,Z 617.702,A -85,B 0,C 180,E1 -29418.39,E2 -29418.39} C_VEL
LIN {X 0,Y 64.39,Z 616.992,A -85,B 0,C 180,E1 -29410.885,E2 -29410.885} C_VEL
LIN {X 0,Y 58.86,Z 614.857,A -85,B 0,C 180,E1 -29396.693,E2 -29396.693} C_VEL
LIN {X 0,Y 57.622,Z 612.917,A -85,B 0,C 180,E1 -29387.032,E2 -29387.032} C_VEL
LIN {X 0,Y 53.641,Z 614.232,A -85,B 0,C 180,E1 -29389.071,E2 -29389.071} C_VEL
LIN {X 0,Y 44.356,Z 617.591,A -85,B 0,C 180,E1 -29401.616,E2 -29401.616} C_VEL
LIN {X 0,Y 38.111,Z 619.142,A -85,B 0,C 180,E1 -29419.37,E2 -29419.37} C_VEL
LIN {X 0,Y 36.859,Z 619.436,A -85,B 0,C 180,E1 -29429.997,E2 -29429.997} C_VEL
LIN {X 0,Y 37.172,Z 619.327,A -85,B 0,C 180,E1 -29434.028,E2 -29434.028} C_VEL
LIN {X 0,Y 39.133,Z 619.088,A -85,B 0,C 180,E1 -29441.376,E2 -29441.376} C_VEL
LIN {X 0,Y 42.637,Z 618.699,A -85,B 0,C 180,E1 -29446.984,E2 -29446.984} C_VEL
LIN {X 0,Y 51.227,Z 617.275,A -85,B 0,C 180,E1 -29454.984,E2 -29454.984} C_VEL
LIN {X 0,Y 53.377,Z 616.753,A -85,B 0,C 180,E1 -29456.741,E2 -29456.741} C_VEL
LIN {X 0,Y 59.744,Z 617.987,A -85,B 0,C 180,E1 -29443.605,E2 -29443.605} C_VEL
LIN {X 0,Y 70.33,Z 618.423,A -85,B 0,C 180,E1 -29432.239,E2 -29432.239} C_VEL
LIN {X 0,Y 73.269,Z 618.435,A -85,B 0,C 180,E1 -29429.998,E2 -29429.998} C_VEL
LIN {X 0,Y 63.916,Z 618.341,A -85,B 0,C 180,E1 -29421.708,E2 -29421.708} C_VEL
LIN {X 0,Y 54.123,Z 617.023,A -85,B 0,C 180,E1 -29405.352,E2 -29405.352} C_VEL
LIN {X 0,Y 53.38,Z 616.752,A -85,B 0,C 180,E1 -29403.258,E2 -29403.258} C_VEL
LIN {X 0,Y 50.738,Z 617.396,A -85,B 0,C 180,E1 -29405.444,E2 -29405.444} C_VEL
LIN {X 0,Y 45.117,Z 618.947,A -85,B 0,C 180,E1 -29421.036,E2 -29421.036} C_VEL
LIN {X 0,Y 43.955,Z 619.241,A -85,B 0,C 180,E1 -29429.997,E2 -29429.997} C_VEL
LIN {X 0,Y 47.468,Z 618.337,A -85,B 0,C 180,E1 -29447.222,E2 -29447.222} C_VEL
LIN {X 0,Y 50.733,Z 617.396,A -85,B 0,C 180,E1 -29454.553,E2 -29454.553} C_VEL
LIN {X 0,Y 51.227,Z 617.275,A -85,B 0,C 180,E1 -29454.984,E2 -29454.984} C_VEL
LIN {X 0,Y 52.166,Z 617.216,A -85,B 0,C 180,E1 -29454.829,E2 -29454.829} C_VEL
LIN {X 0,Y 53.357,Z 617.348,A -85,B 0,C 180,E1 -29453.035,E2 -29453.035} C_VEL
LIN {X 0,Y 54.382,Z 617.786,A -85,B 0,C 180,E1 -29448.202,E2 -29448.202} C_VEL
LIN {X 0,Y 55.827,Z 618.627,A -85,B 0,C 180,E1 -29438.721,E2 -29438.721} C_VEL
LIN {X 0,Y 57.935,Z 618.683,A -85,B 0,C 180,E1 -29434.679,E2 -29434.679} C_VEL
LIN {X 0,Y 58.525,Z 618.685,A -85,B 0,C 180,E1 -29434.002,E2 -29434.002} C_VEL
LIN {X 0,Y 62.788,Z 618.723,A -85,B 0,C 180,E1 -29429.998,E2 -29429.998} C_VEL
LIN {X 0,Y 54.167,Z 618.632,A -85,B 0,C 180,E1 -29420.782,E2 -29420.782} C_VEL
LIN {X 0,Y 52.183,Z 618.751,A -85,B 0,C 180,E1 -29422.258,E2 -29422.258} C_VEL
LIN {X 0,Y 51.077,Z 619.045,A -85,B 0,C 180,E1 -29429.998,E2 -29429.998} C_VEL
LIN {X 0,Y 52.179,Z 618.751,A -85,B 0,C 180,E1 -29437.738,E2 -29437.738} C_VEL
LIN {X 0,Y 54.165,Z 618.632,A -85,B 0,C 180,E1 -29439.225,E2 -29439.225} C_VEL
LIN {X 0,Y 58.525,Z 618.685,A -85,B 0,C 180,E1 -29434.002,E2 -29434.002} C_VEL
LIN {X 0,Y 58.525,Z 618.685,A -85,B 0,C 180,E1 -29434.002,E2 -29434.002}

QRS_NEXT_CUT()

QRS_NEXT()
QRS_HOME()

END
